PROGRAM P_Serial
VAR
END_VAR

P_EL600x();
P_LEDstatus();
P_SerialRemote();
P_JoystickSetup();

END_PROGRAM

(* stored: Version 1.1.0.1, ProductVersion 3.1.4022.3
   POU P_Serial: Id {012e2640-da2b-48e3-a4a8-f6b320642620}, SpecialFunc None *)
